KUKA KRL program: ConnectFour.src, ConnectFour.dat

--- ConnectFour.src ---
&ACCESS RVP
&REL 8
&PARAM DISKPATH = KRC:\R1\Program

DEF ConnectFour()

    ; Initialize robot motion system
    BAS(#initmov,0)

    ; Select tool
    BAS(#tool,3)

    ; Select base coordinate
    BAS(#base,3)

    ; Move robot to its current axis position
    PTP $AXIS_ACT
    p_start = $nullframe

    CELL_SEL = -1
    SYNC_VAR = 1

    LOOP

        mod_assert = modulo(SYNC_VAR, 2)
        IF (mod_assert == 0) THEN

            IF (CELL_SEL >= 1) AND (CELL_SEL <= (cols*rows)) THEN

                ; Convert linear cell number to row and column
                cell_num = CELL_SEL
                row = (cell_num - 1) / cols + 1
                col = modulo((cell_num - 1), cols) + 1

                ; Draw an X in the selected cell
                DrawCross()

                ; Reset cell selection
                reset_vars = 1

            ENDIF

            IF (CELL_SEL == 0) THEN

                ; Draw Connect Four board
                DrawBoard()

                ; Reset cell selection
                reset_vars = 1

            ENDIF

        ENDIF

        WAIT SEC 0.8

        ; Move to a waiting position
        PTP {X -49.67, Y 11.9, Z 261.33, A 0, B 0, C 0, S 2, T 3}

	IF (reset_vars == 1) THEN
		; Reset cell selection
                CELL_SEL = -1
                SYNC_VAR = SYNC_VAR + 1
		reset_vars = 0
	ENDIF


    ENDLOOP

END


DEF DrawBoard()

    ; Compute overall board dimensions
    board_width  = cols * cell_size
    board_height = rows * cell_size

    ; Draw vertical grid lines (cols - 1 lines)
    idx = 1
    LOOP
        IF idx > (cols - 1) THEN
            EXIT
        ENDIF

        ; Move above start
        pos0 = p_start
        pos0.X = (origin_x + idx * cell_size)
        pos0.Y = origin_y
        pos0.Z = z_safe
        PTP pos0

        ; Lower tool to drawing height
        pos0.Z = z_draw
        LIN pos0

        ; Draw vertical line upward
        pos0.Y = origin_y + board_height
        LIN pos0

        ; Lift tool back to safe height
        pos0.Z = z_safe
        PTP pos0

        idx = idx + 1
    ENDLOOP


    ; Draw horizontal grid lines (rows - 1 lines)
    idx = 1
    LOOP
        IF idx > (rows - 1) THEN
            EXIT
        ENDIF

        ; Move above start
        pos0 = p_start
        pos0.X = origin_x
        pos0.Y = (origin_y + idx * cell_size)
        pos0.Z = z_safe
        PTP pos0

        ; Lower tool to drawing height
        pos0.Z = z_draw
        LIN pos0

        ; Draw horizontal line to the right
        pos0.X = origin_x + board_width
        LIN pos0

        ; Lift tool back to safe height
        pos0.Z = z_safe
        PTP pos0

        idx = idx + 1
    ENDLOOP

    ; Draw outer frame (quick implementation)
    pos0 = $nullframe
    pos0.Z = z_safe
    PTP pos0

    pos0.Z = z_draw
    LIN pos0

    pos0.X = cell_size * 6
    LIN pos0

    pos0.Y = cell_size * 7
    LIN pos0

    pos0.X = 0
    LIN pos0

    pos0.Y = 0
    LIN pos0

    LIN {Z 10}
END


DEF DrawCross()

    ; calculate center of selected cell
    cx = origin_x + (col - 1) * cell_size + cell_size / 2
    cy = origin_y + (row - 1) * cell_size + cell_size / 2
    r = cell_size / 3

    ; First diagonal
    pos1 = p_start
    pos1.X = (cx - r)
    pos1.Y = (cy - r)
    pos1.Z = z_safe

    pos2 = p_start
    pos2.X = (cx + r)
    pos2.Y = (cy + r)
    pos2.Z = z_draw

    ; Move above start point
    PTP pos1

    ; Lower pen and draw diagonal
    pos1.Z = z_draw
    LIN pos1
    LIN pos2

    ; Lift pen
    pos2.Z = z_safe
    PTP pos2

    ; Second diagonal
    pos1 = p_start
    pos1.X = (cx - r)
    pos1.Y = (cy + r)
    pos1.Z = z_safe

    pos2 = p_start
    pos2.X = (cx + r)
    pos2.Y = (cy - r)
    pos2.Z = z_draw

    ; Move above start point
    PTP pos1

    ; Lower pen and draw diagonal
    pos1.Z = z_draw
    LIN pos1
    LIN pos2

    ; Lift pen
    pos2.Z = z_safe
    PTP pos2
END


DEFFCT INT modulo(mod_arg_a:IN, mod_arg_b:IN)

    DECL INT mod_arg_a
    DECL INT mod_arg_b

    return (mod_arg_a - mod_arg_b * (mod_arg_a / mod_arg_b))

ENDFCT

--- ConnectFour.dat ---
&ACCESS RVP
&REL 8
&PARAM DISKPATH = KRC:\R1\Program
DEFDAT  connectfour

;; ------------------------------------------------------------------
;; api related variables:
;;
;; SYNC_VAR: Synchronization variable for communication between robot and computer
;;
;; - Even value  : Robot is allowed to execute its task
;;                 After finishing, the robot increments SYNC_VAR by 1
;; - Odd value   : Robot waits. Computer may read/write commands
;;                 Computer increments SYNC_VAR by 1 when ready
;;
;; CELL_SEL: Cell selection command variable
;;
;; - Default value: -1 (No action)
;; - Value 0      : Draw the game field
;; - Value 1..42  : Draw a cross in the selected cell (cell index mapping predefined)
;;
;; Notice !!!
;;    Both lines must be placed in config file
;;    INT CELL_SEL = -1
;;    INT SYNC_VAR = 0
;; ------------------------------------------------------------------

; the game field origin position
DECL REAL origin_x=0.0
DECL REAL origin_y=0.0

; drawing height and safe clearance height
DECL REAL z_draw=-16.0000
DECL REAL z_safe=5.00000

; modulo assertion
INT mod_assert=1

; the return value of modulo function
DECL INT mod_result

; number of colomns and rows of the game field
DECL INT cols=6
DECL INT rows=7

; game field attributes
DECL INT row
DECL INT col
DECL INT cell_num
DECL REAL board_width
DECL REAL board_height

; cell width and height
DECL REAL cell_size=10.00000

; cell center coordinate
DECL REAL cx
DECL REAL cy
DECL REAL r

; variables to draw the game field
DECL FRAME pos0
DECL FRAME pos1
DECL FRAME pos2
DECL FRAME p_start

; iteration variable
DECL INT idx

; controll reset block
DECL INT reset_vars = 0

ENDDAT
